PROGRAM MAIN
VAR
	//bInput1 AT %I*: BOOL;
	//bOutput2 AT %Q*:BOOL;
	bBackhofengedruckt :BOOL;
	Sfertig AT %Q* :BOOL;
	fbtimer AT %I* :TP;
	fbtrigger :R_TRIG;
	Anzahlpizza:DINT;
	testBit:BOOL;
Temperatur AT %I*: INT;
angezeigterWert:LREAL;
angezeigterWert1:INT;
angezeigterWert2:REAL;
Temperatureanzeige:STRING;





	
	
END_VAR

//bOutput2:=NOT bInput1;
angezeigterWert:=INT_TO_REAL(Temperatur)/100;
//angezeigterWert1:=REAL_TO_INT(angezeigterWert*100);
//angezeigterWert2:=INT_TO_REAL(angezeigterWert1/100);
temperatureanzeige:=LREAL_TO_FMTSTR(angezeigterWert, 2, TRUE);
	
	
fbtimer(IN:=bBackhofengedruckt, PT:=T#5S);
	Sfertig:=fbtimer.Q;
fbtrigger(clk:=Sfertig);
IF fbtrigger.Q THEN
	Anzahlpizza:= Anzahlpizza+1;
	//angezeigterWert:=INT_TO_REAL(Temperatur)/100;
	//angezeigterWert:= temperatur/100;
	
END_IF

pou();

END_PROGRAM

(* stored: Version 1.1.0.1, ProductVersion 3.1.4024.4
   POU MAIN: Id {ae65c23e-b8e6-408d-9d93-fb7e9005409a}, SpecialFunc None *)
